TYPE ST_HardwareConfigure_DB :
STRUCT
	iParametersID			: INT;
	wsConfigureItem			: WSTRING(255);
	wsConfigureName			: WSTRING(255);
	wsConfigureValue		: WSTRING(255);
	wsDataType				: WSTRING(255);
	wsDescription			: WSTRING(255);
END_STRUCT
END_TYPE

(* stored: Version 1.1.0.1, ProductVersion 3.1.4024.11
   DUT ST_HardwareConfigure_DB: Id {bf6503d3-3a09-46a3-b3ba-e8694e222031} *)
